TYPE ST_SAFETY_FBAND:
STRUCT
	uStatus							: U_SAFETY_AND; 		(* Typ zalezny od bloku *)
	eState							: E_SAFETY_FBState;		(* Enum ze statusem bloku *)
	bGeneralError					: BOOL; 				(* Gdy wystapi chociaz jeden Error *)
END_STRUCT
END_TYPE

(* stored: Version 1.1.0.1, ProductVersion 3.1.4022.12
   DUT ST_SAFETY_FBAND: Id {166f0ac0-7ff3-402c-af2d-865b7c843f33} *)
